// TIA Portal V18 export
FUNCTION "ST10_Warning" : Void   // FC1006, LAD
{ S7_Optimized_Access := 'FALSE' }
// stored: AutoNumber false, SetENOAutomatically false
   VAR_TEMP
      tpAlwayoff : Bool;
   END_VAR
BEGIN

REGION Network 1
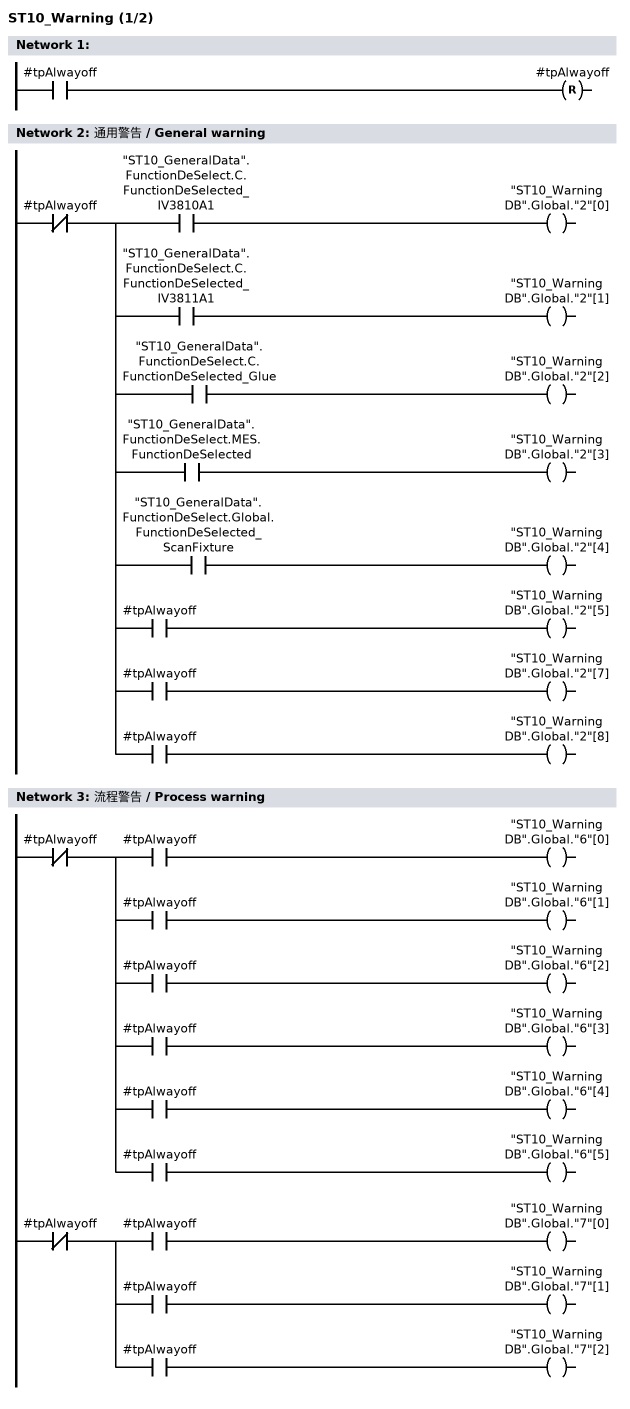
   RUNG wire#powerrail
      Contact( #tpAlwayoff )
      R_Coil( #tpAlwayoff )
   END_RUNG
   // the same network as SCL:
   IF #tpAlwayoff THEN #tpAlwayoff := FALSE; END_IF;
END_REGION

REGION Network 2: 通用警告 / General warning
   RUNG wire#powerrail
      I_Contact( #tpAlwayoff )
      wire#w1
      Contact( "ST10_GeneralData".FunctionDeSelect.C.FunctionDeSelected_IV3810A1 )
      Coil( "ST10_WarningDB".Global."2"[0] )
   END_RUNG
   RUNG wire#w1
      Contact( "ST10_GeneralData".FunctionDeSelect.C.FunctionDeSelected_IV3811A1 )
      Coil( "ST10_WarningDB".Global."2"[1] )
   END_RUNG
   RUNG wire#w1
      Contact( "ST10_GeneralData".FunctionDeSelect.C.FunctionDeSelected_Glue )
      Coil( "ST10_WarningDB".Global."2"[2] )
   END_RUNG
   RUNG wire#w1
      Contact( "ST10_GeneralData".FunctionDeSelect.MES.FunctionDeSelected )
      Coil( "ST10_WarningDB".Global."2"[3] )
   END_RUNG
   RUNG wire#w1
      Contact( "ST10_GeneralData".FunctionDeSelect.Global.FunctionDeSelected_ScanFixture )
      Coil( "ST10_WarningDB".Global."2"[4] )
   END_RUNG
   RUNG wire#w1
      Contact( #tpAlwayoff )
      Coil( "ST10_WarningDB".Global."2"[5] )
   END_RUNG
   RUNG wire#w1
      Contact( #tpAlwayoff )
      Coil( "ST10_WarningDB".Global."2"[7] )
   END_RUNG
   RUNG wire#w1
      Contact( #tpAlwayoff )
      Coil( "ST10_WarningDB".Global."2"[8] )
   END_RUNG
   // the same network as SCL:
   "ST10_WarningDB".Global."2"[0] := NOT #tpAlwayoff AND "ST10_GeneralData".FunctionDeSelect.C.FunctionDeSelected_IV3810A1;
   "ST10_WarningDB".Global."2"[1] := NOT #tpAlwayoff AND "ST10_GeneralData".FunctionDeSelect.C.FunctionDeSelected_IV3811A1;
   "ST10_WarningDB".Global."2"[2] := NOT #tpAlwayoff AND "ST10_GeneralData".FunctionDeSelect.C.FunctionDeSelected_Glue;
   "ST10_WarningDB".Global."2"[3] := NOT #tpAlwayoff AND "ST10_GeneralData".FunctionDeSelect.MES.FunctionDeSelected;
   "ST10_WarningDB".Global."2"[4] := NOT #tpAlwayoff AND "ST10_GeneralData".FunctionDeSelect.Global.FunctionDeSelected_ScanFixture;
   "ST10_WarningDB".Global."2"[5] := NOT #tpAlwayoff AND #tpAlwayoff;
   "ST10_WarningDB".Global."2"[7] := NOT #tpAlwayoff AND #tpAlwayoff;
   "ST10_WarningDB".Global."2"[8] := NOT #tpAlwayoff AND #tpAlwayoff;
END_REGION

REGION Network 3: 流程警告 / Process warning
   RUNG wire#powerrail
      I_Contact( #tpAlwayoff )
      wire#w1
      Contact( #tpAlwayoff )
      Coil( "ST10_WarningDB".Global."6"[0] )
   END_RUNG
   RUNG wire#w1
      Contact( #tpAlwayoff )
      Coil( "ST10_WarningDB".Global."6"[1] )
   END_RUNG
   RUNG wire#w1
      Contact( #tpAlwayoff )
      Coil( "ST10_WarningDB".Global."6"[2] )
   END_RUNG
   RUNG wire#w1
      Contact( #tpAlwayoff )
      Coil( "ST10_WarningDB".Global."6"[3] )
   END_RUNG
   RUNG wire#w1
      Contact( #tpAlwayoff )
      Coil( "ST10_WarningDB".Global."6"[4] )
   END_RUNG
   RUNG wire#w1
      Contact( #tpAlwayoff )
      Coil( "ST10_WarningDB".Global."6"[5] )
   END_RUNG
   RUNG wire#powerrail
      I_Contact( #tpAlwayoff )
      wire#w2
      Contact( #tpAlwayoff )
      Coil( "ST10_WarningDB".Global."7"[0] )
   END_RUNG
   RUNG wire#w2
      Contact( #tpAlwayoff )
      Coil( "ST10_WarningDB".Global."7"[1] )
   END_RUNG
   RUNG wire#w2
      Contact( #tpAlwayoff )
      Coil( "ST10_WarningDB".Global."7"[2] )
   END_RUNG
   // the same network as SCL:
   "ST10_WarningDB".Global."6"[0] := NOT #tpAlwayoff AND #tpAlwayoff;
   "ST10_WarningDB".Global."6"[1] := NOT #tpAlwayoff AND #tpAlwayoff;
   "ST10_WarningDB".Global."6"[2] := NOT #tpAlwayoff AND #tpAlwayoff;
   "ST10_WarningDB".Global."6"[3] := NOT #tpAlwayoff AND #tpAlwayoff;
   "ST10_WarningDB".Global."6"[4] := NOT #tpAlwayoff AND #tpAlwayoff;
   "ST10_WarningDB".Global."6"[5] := NOT #tpAlwayoff AND #tpAlwayoff;
   "ST10_WarningDB".Global."7"[0] := NOT #tpAlwayoff AND #tpAlwayoff;
   "ST10_WarningDB".Global."7"[1] := NOT #tpAlwayoff AND #tpAlwayoff;
   "ST10_WarningDB".Global."7"[2] := NOT #tpAlwayoff AND #tpAlwayoff;
END_REGION

REGION Network 4: 标定警告 / Calibration warning
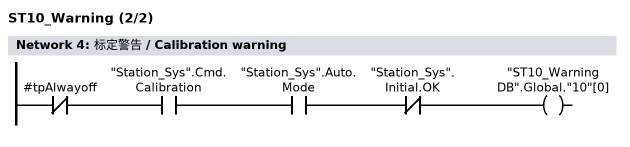
   RUNG wire#powerrail
      I_Contact( #tpAlwayoff )
      Contact( "Station_Sys".Cmd.Calibration )
      Contact( "Station_Sys".Auto.Mode )
      I_Contact( "Station_Sys".Initial.OK )
      Coil( "ST10_WarningDB".Global."10"[0] )
   END_RUNG
   // the same network as SCL:
   "ST10_WarningDB".Global."10"[0] := NOT #tpAlwayoff AND "Station_Sys".Cmd.Calibration AND "Station_Sys".Auto.Mode AND NOT "Station_Sys".Initial.OK;
END_REGION
END_FUNCTION
